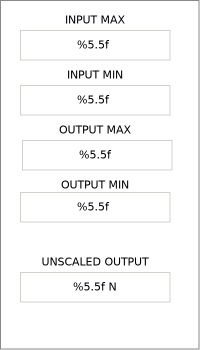
VISUALIZATION VISU_WORD_TO_BYTES  // 200x350
VAR_IN_OUT
	fbVISU:				FB_VISU_WORD_TO_BYTES;
END_VAR
    Textfield (20,30 150x30), "%5.5f", text variable: fbVISU.lrXMax
        OnMouseClick: write the text variable via Default, min 0, max 16085
    Label (20,5 150x30), "INPUT MAX"
    Textfield (20,85 150x30), "%5.5f", text variable: fbVISU.lrXMin
        OnMouseClick: write the text variable via Default, min 0, max 16085
    Label (20,60 150x30), "INPUT MIN"
    Textfield (22,140 150x30), "%5.5f", text variable: fbVISU.lrYMax
        OnMouseClick: write the text variable via Default, min 0
    Label (20,115 150x30), "OUTPUT MAX"
    Textfield (20,192 150x30), "%5.5f", text variable: fbVISU.lrYMin
        OnMouseClick: write the text variable via Default, min 0
    Label (20,170 150x30), "OUTPUT MIN"
    Textfield (20,272 150x30), "%5.5f N", text variable: fbVISU.lrUnscaledInput
        OnMouseClick: write the text variable via Default, min 0
    Label (20,247 150x30), "UNSCALED OUTPUT"
END_VISUALIZATION

(* stored: Version 1.1.0.1, ProductVersion 3.1.4024.9
   Visu VISU_WORD_TO_BYTES: Id {4584404a-e3e2-4900-8deb-89bcf08b40a0} *)
